# B&R Automation Studio project AsProject
Automation Studio 6.5.1.7

## Configuration Config1

CPU X20CP1685, AutomationRuntime 6.4.2, Build 11.3.0

### Task classes (Cpu.sw)
```
Cyclic#4:
  Main <- Main.prg
```

### Hardware
```
X20CP1685 : X20CP1685 v1.9.0.0
  FileDevice1
  FileDeviceName1 = USER
  FileDevicePath1 = USER_PATH
```

## Logical view

### Program Logical/Main (IEC)

#### Cyclic.st
```iecst
PROGRAM _CYCLIC
	(* Insert code here *)
	 (* tässä muutos *)
END_PROGRAM
```

### Program Logical/Program (IEC)

#### Variables.var
```iecst
VAR
	value : INT;
END_VAR
```

#### Cyclic.st
```iecst
PROGRAM _CYCLIC
	(* Insert code here *)

	value := value +1;
	//joo
END_PROGRAM
```

Listed in the project but not available here: Logical/Global.typ, Logical/Global.var, Logical/Libraries
